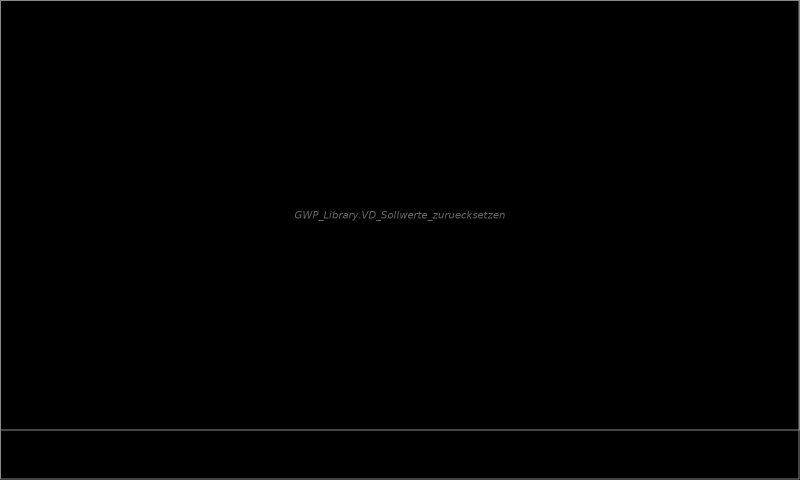
VISUALIZATION VD_Sollwerte_zuruecksetzen  // 800x480
    Frame (0,0 800x430)
        shows GWP_Library.VD_Sollwerte_zuruecksetzen(FB_VD := Main.VD_0, FB_Init_1 := Main.Init_0)
END_VISUALIZATION

(* stored: Version 1.1.0.1, ProductVersion 3.1.4022.6
   Visu VD_Sollwerte_zuruecksetzen: Id {028d0474-d0ce-4787-9df1-a000c32e61d3} *)
